// TIA Portal V18 export
DATA_BLOCK "AHUDelays"   // DB110
{ S7_Optimized_Access := 'FALSE' }
VERSION : 0.1
// stored: AutoNumber false, DBAccessibleFromOPCUA true, IsOnlyStoredInLoadMemory false, IsWriteProtectedInAS false
   VAR RETAIN
      DelaysForStatus { S7_SetPoint := 'True'} : "UDT_AHUsStsDelay";
   END_VAR
BEGIN
END_DATA_BLOCK
